// TIA Portal V17 export
// export: Created 2025-03-05T08:02:46.8342554Z, ExportSetting WithDefaults, DisplayName Totally Integrated Automation Portal, DisplayVersion V17 Update 8, DisplayName TIA Portal Openness, DisplayVersion V17 Update 8, DisplayName TIA Portal Version Control Interface, DisplayVersion V17, DisplayName SINAMICS Startdrive Advanced, DisplayVersion V17 SP2, DisplayName SINAMICS Startdrive G110M, G120, G120C, G120D, G120P, G115D, DisplayVersion V17 SP2, DisplayName SINAMICS Startdrive G130, G150, S120, S150, SINAMICS MV, S210, DisplayVersion V17 SP2, DisplayName STEP 7 Professional, DisplayVersion V17 Update 8, DisplayName SINUMERIK ONE STEP 7 Toolbox, DisplayVersion V17 Update 12, DisplayName SINUMERIK 840D sl STEP 7 Toolbox, DisplayVersion V17 Update 12, DisplayName STEP 7 Safety, DisplayVersion V17 Update 6, DisplayName WinCC Advanced, DisplayVersion V17 Update 8
FUNCTION "FC2120_MPP_ITC_IPC" : Void   // FC2120, LAD
{ S7_Optimized_Access := 'FALSE' }
AUTHOR : ETXETAR
VERSION : 1.0
// stored: AutoNumber false, IsIECCheckEnabled false, SetENOAutomatically false, UDAEnableTagReadback false
   VAR_TEMP
      O_BYTE_0 : Struct   // OPTIONS BYTE 0
         IPC : Bool;   // IPC OPTION
      END_STRUCT;
      TCU_INDEX_SEL : Int;
   END_VAR
   VAR CONSTANT
      FC_NUMBER : DInt := 2120;   // FC NUMBER
   END_VAR
   VAR_TEMP   // added for the SCL form of the ladder/FBD networks
      _w1 : Bool;
      _w2 : Bool;
   END_VAR
BEGIN

REGION Network 1: OPTIONS
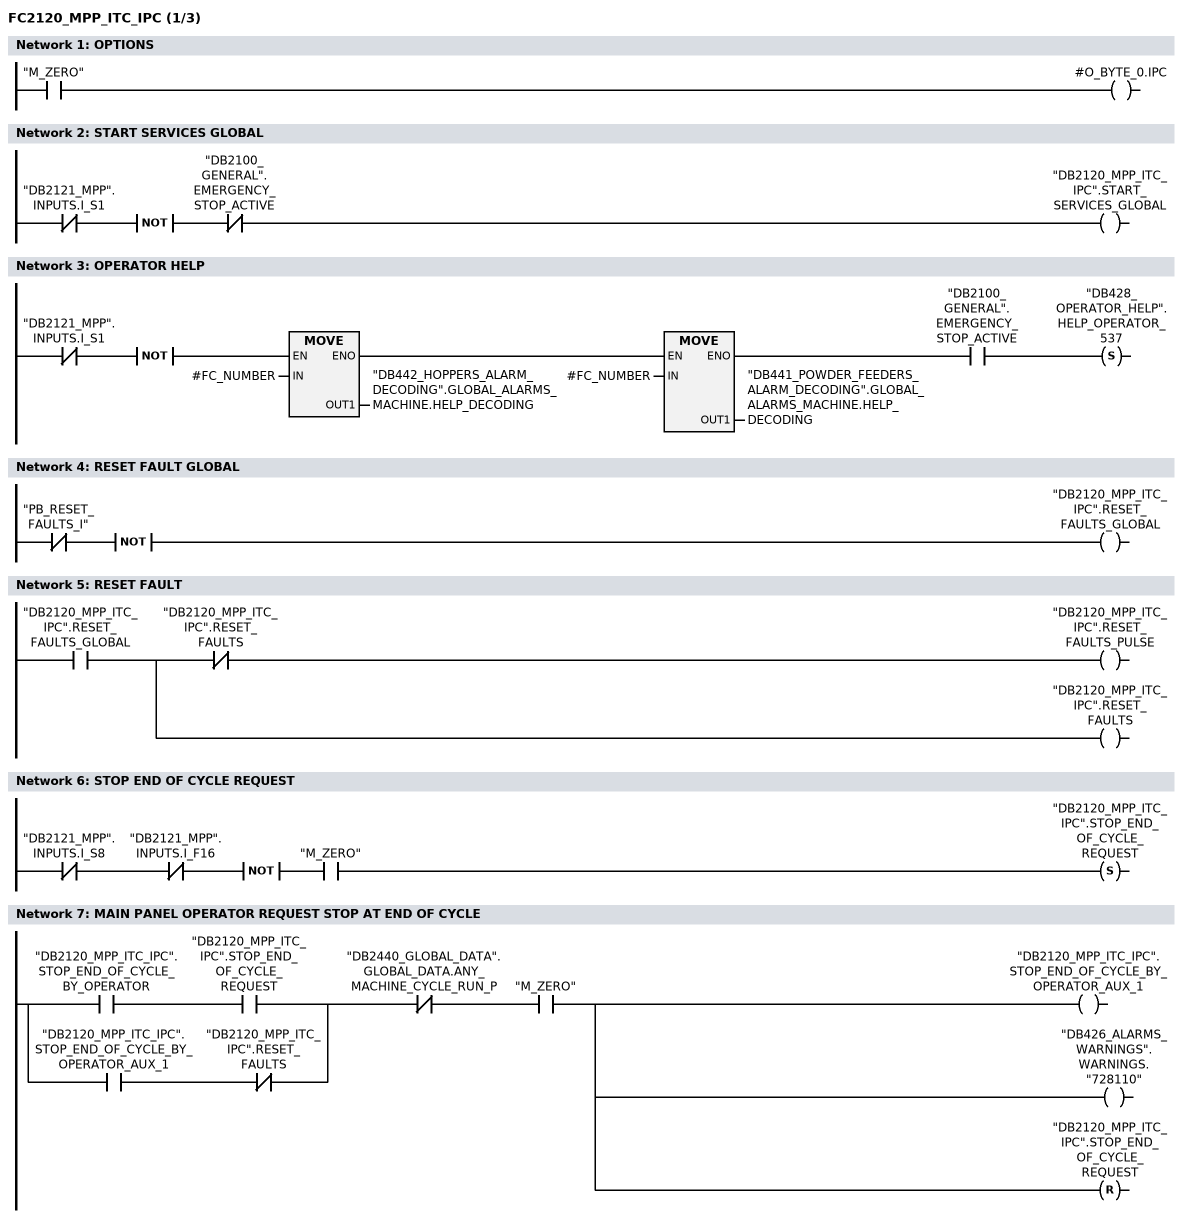
   RUNG wire#powerrail
      Contact( "M_ZERO" )
      Coil( #O_BYTE_0.IPC )
   END_RUNG
   // the same network as SCL:
   #O_BYTE_0.IPC := "M_ZERO";
END_REGION

REGION Network 2: START SERVICES GLOBAL
   RUNG wire#powerrail
      I_Contact( "DB2121_MPP".INPUTS.I_S1 )
      Not()
      I_Contact( "DB2100_GENERAL".EMERGENCY_STOP_ACTIVE )
      Coil( "DB2120_MPP_ITC_IPC".START_SERVICES_GLOBAL )
   END_RUNG
   // the same network as SCL:
   "DB2120_MPP_ITC_IPC".START_SERVICES_GLOBAL := NOT (NOT "DB2121_MPP".INPUTS.I_S1) AND NOT "DB2100_GENERAL".EMERGENCY_STOP_ACTIVE;
END_REGION

REGION Network 3: OPERATOR HELP
   RUNG wire#powerrail
      I_Contact( "DB2121_MPP".INPUTS.I_S1 )
      Not()
      { S7_GenerateENO := "TRUE" } Move(in := #FC_NUMBER, out1 => "DB442_HOPPERS_ALARM_DECODING".GLOBAL_ALARMS_MACHINE.HELP_DECODING)
      { S7_GenerateENO := "TRUE" } Move(in := #FC_NUMBER, out1 => "DB441_POWDER_FEEDERS_ALARM_DECODING".GLOBAL_ALARMS_MACHINE.HELP_DECODING)
      Contact( "DB2100_GENERAL".EMERGENCY_STOP_ACTIVE )
      S_Coil( "DB428_OPERATOR_HELP".HELP_OPERATOR_537 )
   END_RUNG
   // the same network as SCL:
   // ENO of a box is taken as its EN; it also drops when the box reports an error
   #_w1 := NOT (NOT "DB2121_MPP".INPUTS.I_S1);
   IF #_w1 THEN
       "DB442_HOPPERS_ALARM_DECODING".GLOBAL_ALARMS_MACHINE.HELP_DECODING := #FC_NUMBER;
       "DB441_POWDER_FEEDERS_ALARM_DECODING".GLOBAL_ALARMS_MACHINE.HELP_DECODING := #FC_NUMBER;
   END_IF;
   IF #_w1 AND "DB2100_GENERAL".EMERGENCY_STOP_ACTIVE THEN
       "DB428_OPERATOR_HELP".HELP_OPERATOR_537 := TRUE;
   END_IF;
END_REGION

REGION Network 4: RESET FAULT GLOBAL
   RUNG wire#powerrail
      I_Contact( "PB_RESET_FAULTS_I" )
      Not()
      Coil( "DB2120_MPP_ITC_IPC".RESET_FAULTS_GLOBAL )
   END_RUNG
   // the same network as SCL:
   "DB2120_MPP_ITC_IPC".RESET_FAULTS_GLOBAL := NOT (NOT "PB_RESET_FAULTS_I");
END_REGION

REGION Network 5: RESET FAULT
   RUNG wire#powerrail
      Contact( "DB2120_MPP_ITC_IPC".RESET_FAULTS_GLOBAL )
      wire#w1
      I_Contact( "DB2120_MPP_ITC_IPC".RESET_FAULTS )
      Coil( "DB2120_MPP_ITC_IPC".RESET_FAULTS_PULSE )
   END_RUNG
   RUNG wire#w1
      Coil( "DB2120_MPP_ITC_IPC".RESET_FAULTS )
   END_RUNG
   // the same network as SCL:
   "DB2120_MPP_ITC_IPC".RESET_FAULTS_PULSE := "DB2120_MPP_ITC_IPC".RESET_FAULTS_GLOBAL AND NOT "DB2120_MPP_ITC_IPC".RESET_FAULTS;
   "DB2120_MPP_ITC_IPC".RESET_FAULTS := "DB2120_MPP_ITC_IPC".RESET_FAULTS_GLOBAL;
END_REGION

REGION Network 6: STOP END OF CYCLE REQUEST
   RUNG wire#powerrail
      I_Contact( "DB2121_MPP".INPUTS.I_S8 )
      I_Contact( "DB2121_MPP".INPUTS.I_F16 )
      Not()
      Contact( "M_ZERO" )
      S_Coil( "DB2120_MPP_ITC_IPC".STOP_END_OF_CYCLE_REQUEST )
   END_RUNG
   // the same network as SCL:
   IF NOT (NOT "DB2121_MPP".INPUTS.I_S8 AND NOT "DB2121_MPP".INPUTS.I_F16) AND "M_ZERO" THEN
       "DB2120_MPP_ITC_IPC".STOP_END_OF_CYCLE_REQUEST := TRUE;
   END_IF;
END_REGION

REGION Network 7: MAIN PANEL OPERATOR REQUEST STOP AT END OF CYCLE
   RUNG wire#powerrail
      Contact( "DB2120_MPP_ITC_IPC".STOP_END_OF_CYCLE_BY_OPERATOR )
      Contact( "DB2120_MPP_ITC_IPC".STOP_END_OF_CYCLE_REQUEST )
      wire#w1
      I_Contact( "DB2440_GLOBAL_DATA".GLOBAL_DATA.ANY_MACHINE_CYCLE_RUN_P )
      Contact( "M_ZERO" )
      wire#w2
      Coil( "DB2120_MPP_ITC_IPC".STOP_END_OF_CYCLE_BY_OPERATOR_AUX_1 )
   END_RUNG
   RUNG wire#powerrail
      Contact( "DB2120_MPP_ITC_IPC".STOP_END_OF_CYCLE_BY_OPERATOR_AUX_1 )
      I_Contact( "DB2120_MPP_ITC_IPC".RESET_FAULTS )
   END_RUNG wire#w1
   RUNG wire#w2
      Coil( "DB426_ALARMS_WARNINGS".WARNINGS."728110" )
   END_RUNG
   RUNG wire#w2
      R_Coil( "DB2120_MPP_ITC_IPC".STOP_END_OF_CYCLE_REQUEST )
   END_RUNG
   // the same network as SCL:
   "DB2120_MPP_ITC_IPC".STOP_END_OF_CYCLE_BY_OPERATOR_AUX_1 := (("DB2120_MPP_ITC_IPC".STOP_END_OF_CYCLE_BY_OPERATOR AND "DB2120_MPP_ITC_IPC".STOP_END_OF_CYCLE_REQUEST) OR ("DB2120_MPP_ITC_IPC".STOP_END_OF_CYCLE_BY_OPERATOR_AUX_1 AND NOT "DB2120_MPP_ITC_IPC".RESET_FAULTS)) AND NOT "DB2440_GLOBAL_DATA".GLOBAL_DATA.ANY_MACHINE_CYCLE_RUN_P AND "M_ZERO";
   "DB426_ALARMS_WARNINGS".WARNINGS."728110" := "DB2120_MPP_ITC_IPC".STOP_END_OF_CYCLE_BY_OPERATOR_AUX_1;
   IF "DB2120_MPP_ITC_IPC".STOP_END_OF_CYCLE_BY_OPERATOR_AUX_1 THEN
       "DB2120_MPP_ITC_IPC".STOP_END_OF_CYCLE_REQUEST := FALSE;
   END_IF;
END_REGION

REGION Network 8: AUXILIARY PANEL OPERATOR REQUEST STOP AT END OF CYCLE
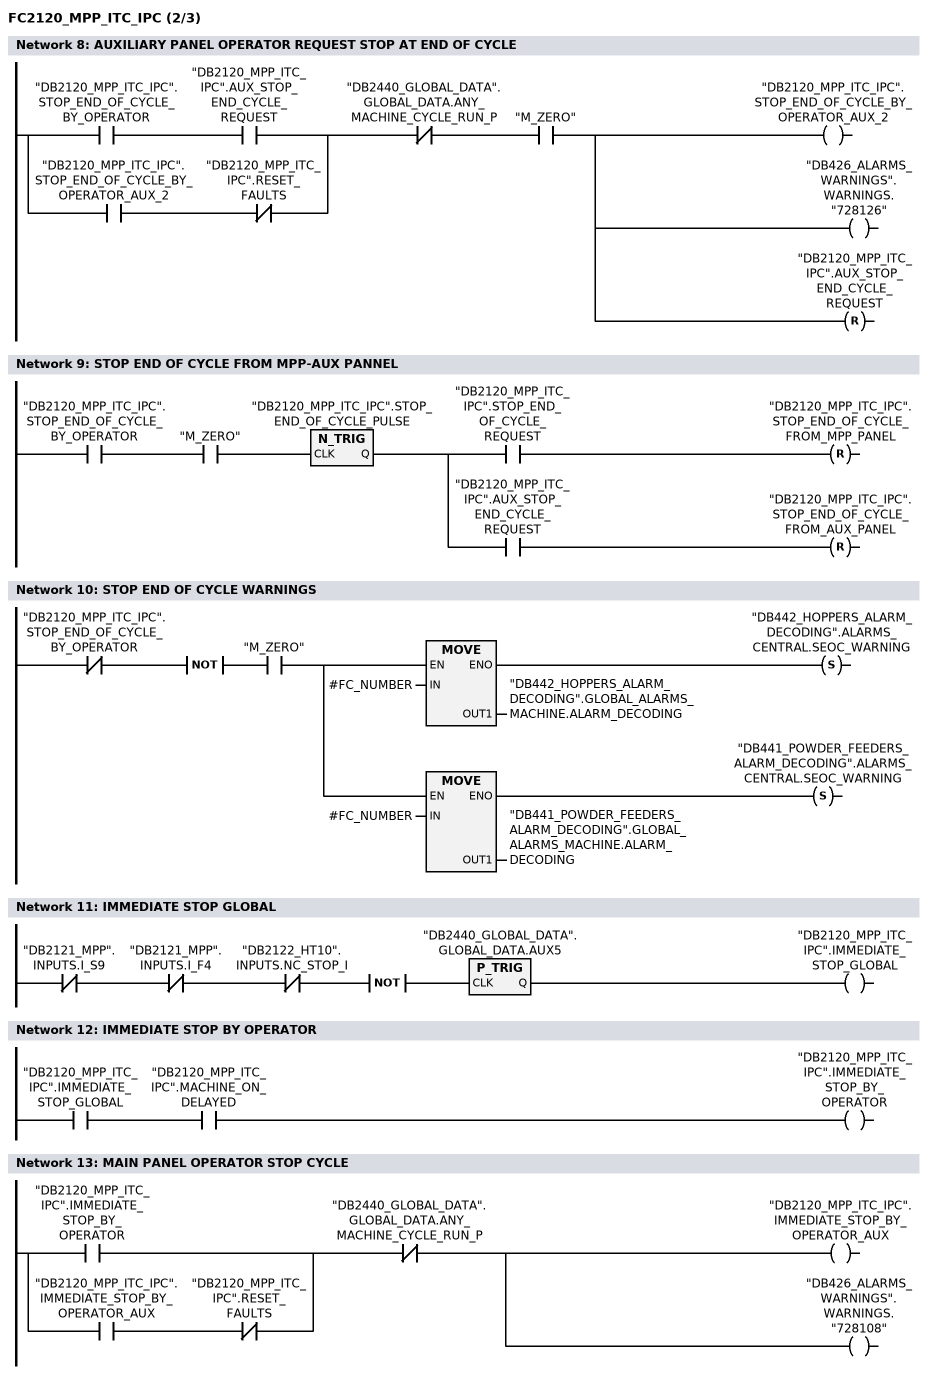
   RUNG wire#powerrail
      Contact( "DB2120_MPP_ITC_IPC".STOP_END_OF_CYCLE_BY_OPERATOR )
      Contact( "DB2120_MPP_ITC_IPC".AUX_STOP_END_CYCLE_REQUEST )
      wire#w1
      I_Contact( "DB2440_GLOBAL_DATA".GLOBAL_DATA.ANY_MACHINE_CYCLE_RUN_P )
      Contact( "M_ZERO" )
      wire#w2
      Coil( "DB2120_MPP_ITC_IPC".STOP_END_OF_CYCLE_BY_OPERATOR_AUX_2 )
   END_RUNG
   RUNG wire#powerrail
      Contact( "DB2120_MPP_ITC_IPC".STOP_END_OF_CYCLE_BY_OPERATOR_AUX_2 )
      I_Contact( "DB2120_MPP_ITC_IPC".RESET_FAULTS )
   END_RUNG wire#w1
   RUNG wire#w2
      Coil( "DB426_ALARMS_WARNINGS".WARNINGS."728126" )
   END_RUNG
   RUNG wire#w2
      R_Coil( "DB2120_MPP_ITC_IPC".AUX_STOP_END_CYCLE_REQUEST )
   END_RUNG
   // the same network as SCL:
   "DB2120_MPP_ITC_IPC".STOP_END_OF_CYCLE_BY_OPERATOR_AUX_2 := (("DB2120_MPP_ITC_IPC".STOP_END_OF_CYCLE_BY_OPERATOR AND "DB2120_MPP_ITC_IPC".AUX_STOP_END_CYCLE_REQUEST) OR ("DB2120_MPP_ITC_IPC".STOP_END_OF_CYCLE_BY_OPERATOR_AUX_2 AND NOT "DB2120_MPP_ITC_IPC".RESET_FAULTS)) AND NOT "DB2440_GLOBAL_DATA".GLOBAL_DATA.ANY_MACHINE_CYCLE_RUN_P AND "M_ZERO";
   "DB426_ALARMS_WARNINGS".WARNINGS."728126" := "DB2120_MPP_ITC_IPC".STOP_END_OF_CYCLE_BY_OPERATOR_AUX_2;
   IF "DB2120_MPP_ITC_IPC".STOP_END_OF_CYCLE_BY_OPERATOR_AUX_2 THEN
       "DB2120_MPP_ITC_IPC".AUX_STOP_END_CYCLE_REQUEST := FALSE;
   END_IF;
END_REGION

REGION Network 9: STOP END OF CYCLE FROM MPP-AUX PANNEL
   RUNG wire#powerrail
      Contact( "DB2120_MPP_ITC_IPC".STOP_END_OF_CYCLE_BY_OPERATOR )
      Contact( "M_ZERO" )
      N_Trig( "DB2120_MPP_ITC_IPC".STOP_END_OF_CYCLE_PULSE )
      wire#w1
      Contact( "DB2120_MPP_ITC_IPC".STOP_END_OF_CYCLE_REQUEST )
      R_Coil( "DB2120_MPP_ITC_IPC".STOP_END_OF_CYCLE_FROM_MPP_PANEL )
   END_RUNG
   RUNG wire#w1
      Contact( "DB2120_MPP_ITC_IPC".AUX_STOP_END_CYCLE_REQUEST )
      R_Coil( "DB2120_MPP_ITC_IPC".STOP_END_OF_CYCLE_FROM_AUX_PANEL )
   END_RUNG
   // the same network as SCL:
   #_w1 := "DB2120_MPP_ITC_IPC".STOP_END_OF_CYCLE_BY_OPERATOR AND "M_ZERO";
   #_w2 := NOT #_w1 AND "DB2120_MPP_ITC_IPC".STOP_END_OF_CYCLE_PULSE;   // falling edge
   "DB2120_MPP_ITC_IPC".STOP_END_OF_CYCLE_PULSE := #_w1;
   IF #_w2 AND "DB2120_MPP_ITC_IPC".STOP_END_OF_CYCLE_REQUEST THEN
       "DB2120_MPP_ITC_IPC".STOP_END_OF_CYCLE_FROM_MPP_PANEL := FALSE;
   END_IF;
   IF #_w2 AND "DB2120_MPP_ITC_IPC".AUX_STOP_END_CYCLE_REQUEST THEN
       "DB2120_MPP_ITC_IPC".STOP_END_OF_CYCLE_FROM_AUX_PANEL := FALSE;
   END_IF;
END_REGION

REGION Network 10: STOP END OF CYCLE WARNINGS
   RUNG wire#powerrail
      I_Contact( "DB2120_MPP_ITC_IPC".STOP_END_OF_CYCLE_BY_OPERATOR )
      Not()
      Contact( "M_ZERO" )
      wire#w1
      { S7_GenerateENO := "TRUE" } Move(in := #FC_NUMBER, out1 => "DB442_HOPPERS_ALARM_DECODING".GLOBAL_ALARMS_MACHINE.ALARM_DECODING)
      S_Coil( "DB442_HOPPERS_ALARM_DECODING".ALARMS_CENTRAL.SEOC_WARNING )
   END_RUNG
   RUNG wire#w1
      { S7_GenerateENO := "TRUE" } Move(in := #FC_NUMBER, out1 => "DB441_POWDER_FEEDERS_ALARM_DECODING".GLOBAL_ALARMS_MACHINE.ALARM_DECODING)
      S_Coil( "DB441_POWDER_FEEDERS_ALARM_DECODING".ALARMS_CENTRAL.SEOC_WARNING )
   END_RUNG
   // the same network as SCL:
   // ENO of a box is taken as its EN; it also drops when the box reports an error
   IF NOT (NOT "DB2120_MPP_ITC_IPC".STOP_END_OF_CYCLE_BY_OPERATOR) AND "M_ZERO" THEN
       "DB442_HOPPERS_ALARM_DECODING".GLOBAL_ALARMS_MACHINE.ALARM_DECODING := #FC_NUMBER;
       "DB442_HOPPERS_ALARM_DECODING".ALARMS_CENTRAL.SEOC_WARNING := TRUE;
       "DB441_POWDER_FEEDERS_ALARM_DECODING".GLOBAL_ALARMS_MACHINE.ALARM_DECODING := #FC_NUMBER;
       "DB441_POWDER_FEEDERS_ALARM_DECODING".ALARMS_CENTRAL.SEOC_WARNING := TRUE;
   END_IF;
END_REGION

REGION Network 11: IMMEDIATE STOP GLOBAL
   RUNG wire#powerrail
      I_Contact( "DB2121_MPP".INPUTS.I_S9 )
      I_Contact( "DB2121_MPP".INPUTS.I_F4 )
      I_Contact( "DB2122_HT10".INPUTS.NC_STOP_I )
      Not()
      P_Trig( "DB2440_GLOBAL_DATA".GLOBAL_DATA.AUX5 )
      Coil( "DB2120_MPP_ITC_IPC".IMMEDIATE_STOP_GLOBAL )
   END_RUNG
   // the same network as SCL:
   #_w1 := NOT (NOT "DB2121_MPP".INPUTS.I_S9 AND NOT "DB2121_MPP".INPUTS.I_F4 AND NOT "DB2122_HT10".INPUTS.NC_STOP_I);
   #_w2 := #_w1 AND NOT "DB2440_GLOBAL_DATA".GLOBAL_DATA.AUX5;   // rising edge
   "DB2440_GLOBAL_DATA".GLOBAL_DATA.AUX5 := #_w1;
   "DB2120_MPP_ITC_IPC".IMMEDIATE_STOP_GLOBAL := #_w2;
END_REGION

REGION Network 12: IMMEDIATE STOP BY OPERATOR
   RUNG wire#powerrail
      Contact( "DB2120_MPP_ITC_IPC".IMMEDIATE_STOP_GLOBAL )
      Contact( "DB2120_MPP_ITC_IPC".MACHINE_ON_DELAYED )
      Coil( "DB2120_MPP_ITC_IPC".IMMEDIATE_STOP_BY_OPERATOR )
   END_RUNG
   // the same network as SCL:
   "DB2120_MPP_ITC_IPC".IMMEDIATE_STOP_BY_OPERATOR := "DB2120_MPP_ITC_IPC".IMMEDIATE_STOP_GLOBAL AND "DB2120_MPP_ITC_IPC".MACHINE_ON_DELAYED;
END_REGION

REGION Network 13: MAIN PANEL OPERATOR STOP CYCLE
   RUNG wire#powerrail
      Contact( "DB2120_MPP_ITC_IPC".IMMEDIATE_STOP_BY_OPERATOR )
      wire#w1
      I_Contact( "DB2440_GLOBAL_DATA".GLOBAL_DATA.ANY_MACHINE_CYCLE_RUN_P )
      wire#w2
      Coil( "DB2120_MPP_ITC_IPC".IMMEDIATE_STOP_BY_OPERATOR_AUX )
   END_RUNG
   RUNG wire#powerrail
      Contact( "DB2120_MPP_ITC_IPC".IMMEDIATE_STOP_BY_OPERATOR_AUX )
      I_Contact( "DB2120_MPP_ITC_IPC".RESET_FAULTS )
   END_RUNG wire#w1
   RUNG wire#w2
      Coil( "DB426_ALARMS_WARNINGS".WARNINGS."728108" )
   END_RUNG
   // the same network as SCL:
   "DB2120_MPP_ITC_IPC".IMMEDIATE_STOP_BY_OPERATOR_AUX := ("DB2120_MPP_ITC_IPC".IMMEDIATE_STOP_BY_OPERATOR OR ("DB2120_MPP_ITC_IPC".IMMEDIATE_STOP_BY_OPERATOR_AUX AND NOT "DB2120_MPP_ITC_IPC".RESET_FAULTS)) AND NOT "DB2440_GLOBAL_DATA".GLOBAL_DATA.ANY_MACHINE_CYCLE_RUN_P;
   "DB426_ALARMS_WARNINGS".WARNINGS."728108" := "DB2120_MPP_ITC_IPC".IMMEDIATE_STOP_BY_OPERATOR_AUX;
END_REGION

REGION Network 14: IMMEDIATE STOP WARNING
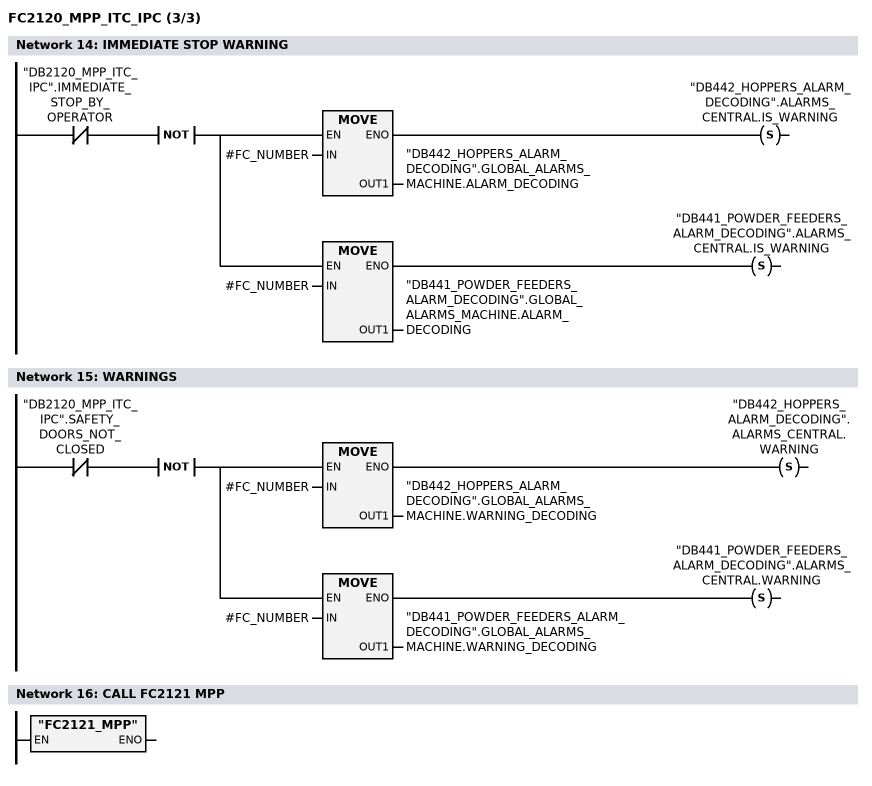
   RUNG wire#powerrail
      I_Contact( "DB2120_MPP_ITC_IPC".IMMEDIATE_STOP_BY_OPERATOR )
      Not()
      wire#w1
      { S7_GenerateENO := "TRUE" } Move(in := #FC_NUMBER, out1 => "DB442_HOPPERS_ALARM_DECODING".GLOBAL_ALARMS_MACHINE.ALARM_DECODING)
      S_Coil( "DB442_HOPPERS_ALARM_DECODING".ALARMS_CENTRAL.IS_WARNING )
   END_RUNG
   RUNG wire#w1
      { S7_GenerateENO := "TRUE" } Move(in := #FC_NUMBER, out1 => "DB441_POWDER_FEEDERS_ALARM_DECODING".GLOBAL_ALARMS_MACHINE.ALARM_DECODING)
      S_Coil( "DB441_POWDER_FEEDERS_ALARM_DECODING".ALARMS_CENTRAL.IS_WARNING )
   END_RUNG
   // the same network as SCL:
   // ENO of a box is taken as its EN; it also drops when the box reports an error
   IF NOT (NOT "DB2120_MPP_ITC_IPC".IMMEDIATE_STOP_BY_OPERATOR) THEN
       "DB442_HOPPERS_ALARM_DECODING".GLOBAL_ALARMS_MACHINE.ALARM_DECODING := #FC_NUMBER;
       "DB442_HOPPERS_ALARM_DECODING".ALARMS_CENTRAL.IS_WARNING := TRUE;
       "DB441_POWDER_FEEDERS_ALARM_DECODING".GLOBAL_ALARMS_MACHINE.ALARM_DECODING := #FC_NUMBER;
       "DB441_POWDER_FEEDERS_ALARM_DECODING".ALARMS_CENTRAL.IS_WARNING := TRUE;
   END_IF;
END_REGION

REGION Network 15: WARNINGS
   RUNG wire#powerrail
      I_Contact( "DB2120_MPP_ITC_IPC".SAFETY_DOORS_NOT_CLOSED )
      Not()
      wire#w1
      { S7_GenerateENO := "TRUE" } Move(in := #FC_NUMBER, out1 => "DB442_HOPPERS_ALARM_DECODING".GLOBAL_ALARMS_MACHINE.WARNING_DECODING)
      S_Coil( "DB442_HOPPERS_ALARM_DECODING".ALARMS_CENTRAL.WARNING )
   END_RUNG
   RUNG wire#w1
      { S7_GenerateENO := "TRUE" } Move(in := #FC_NUMBER, out1 => "DB441_POWDER_FEEDERS_ALARM_DECODING".GLOBAL_ALARMS_MACHINE.WARNING_DECODING)
      S_Coil( "DB441_POWDER_FEEDERS_ALARM_DECODING".ALARMS_CENTRAL.WARNING )
   END_RUNG
   // the same network as SCL:
   // ENO of a box is taken as its EN; it also drops when the box reports an error
   IF NOT (NOT "DB2120_MPP_ITC_IPC".SAFETY_DOORS_NOT_CLOSED) THEN
       "DB442_HOPPERS_ALARM_DECODING".GLOBAL_ALARMS_MACHINE.WARNING_DECODING := #FC_NUMBER;
       "DB442_HOPPERS_ALARM_DECODING".ALARMS_CENTRAL.WARNING := TRUE;
       "DB441_POWDER_FEEDERS_ALARM_DECODING".GLOBAL_ALARMS_MACHINE.WARNING_DECODING := #FC_NUMBER;
       "DB441_POWDER_FEEDERS_ALARM_DECODING".ALARMS_CENTRAL.WARNING := TRUE;
   END_IF;
END_REGION

REGION Network 16: CALL FC2121 MPP
   RUNG wire#powerrail
      "FC2121_MPP"()
   END_RUNG
   // the same network as SCL:
   "FC2121_MPP"();
END_REGION
END_FUNCTION
